{attribute 'no_explicit_call':= 'do not call this POU directly'}
FUNCTION_BLOCK T_Monitor_DINT
VAR
    _CurrentValue  : DINT := UnlikelyValue; 
    _Changed       : BOOL;
END_VAR
VAR CONSTANT
	UnlikelyValue : DINT := 123456789;
END_VAR

PROPERTY Changed : BOOL
GET
Changed := _Changed;
END_GET
END_PROPERTY

METHOD CyclicUpdate : BOOL
VAR_INPUT
    Value : DINT;
END_VAR
_Changed      := Value <> _CurrentValue;
_CurrentValue := Value;
CyclicUpdate  := _Changed;
END_METHOD

METHOD Reset
_CurrentValue := UnlikelyValue;
_Changed      := FALSE;
END_METHOD

END_FUNCTION_BLOCK

(* stored: Version 1.1.0.1, ProductVersion 3.1.4024.12
   POU T_Monitor_DINT: Id {fd5173f9-2778-4890-b57b-bf24b09d715f}, SpecialFunc None
   Folder Methods: Id {316ec2b8-e3f6-407a-94f4-ccb646bf590f}
   Folder Properties: Id {22bb550f-0f2e-4043-90a3-95b56c2f4aac}
   Property Changed: Id {71a14203-c7a9-4b8d-a460-5a9f3565e29b}
   Get Get: Id {c52941b3-e24f-4173-aa8b-8f6c7aff39e5}
   Method CyclicUpdate: Id {c7149b97-608e-4fc4-914f-ba85f35a4193}
   Method Reset: Id {5f291c8f-4dbb-4ae1-9886-c6b6bd429e3e} *)
